(* PLC project RACK2537.project, Inovance company InoProShop(V1.8.1.3) InoProShop(V1.8.1.3) *)
(* stored: creationDateTime 2025-03-21T09:54:46.669365, modificationDateTime 2025-03-07T16:07:54.7010798 *)

TYPE _sDT : STRUCT
  year : DINT;  (* 按360天计算 *)
  month : DINT;  (* 按12个月计算 *)
  day : DINT;  (* 按30天计算 *)
  hour : DINT;  (* 按24小时 *)
  min : DINT;  (* 按60分钟 *)
  sec : DINT;  (* 按60秒 *)
END_STRUCT;
END_TYPE

FUNCTION_BLOCK 累计TIME
  VAR_INPUT
    EN : BOOL;
  END_VAR
  VAR
    心跳 : BOOL;
    TON_0 : TON;
    PLS_0 : PLS;
    TON_1 : TON;
  END_VAR
  VAR_INPUT
    清除 : BOOL;
  END_VAR
  VAR_OUTPUT
    ENO : BOOL;
    累计时间 : DINT;
  END_VAR
  VAR
    转换参数 : _sDT;
  END_VAR
  VAR_OUTPUT
    时间转换 : _sDT;
  END_VAR
  VAR  (* added by the conversion: wires and edge detectors of the diagram *)
    _GT49_ENO : BOOL;
    _GT49_OUT : BOOL;
  END_VAR

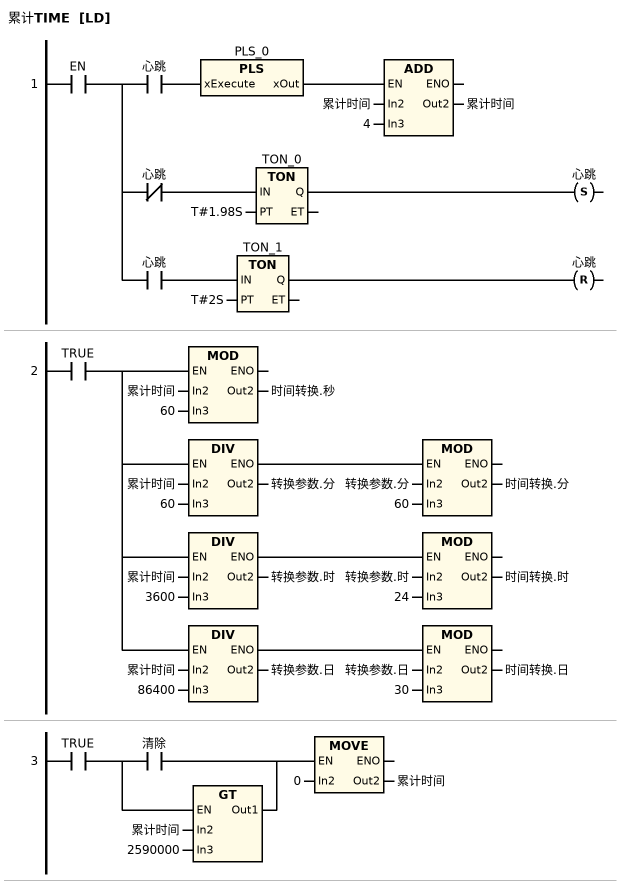
(* LD diagram, written out as Structured Text *)
(* 计时 *)

PLS_0(xExecute := EN AND 心跳);
IF PLS_0.xOut THEN 累计时间 := 累计时间 + 4; END_IF;
TON_0(IN := EN AND NOT 心跳, PT := T#1.98S);
IF TON_0.Q THEN 心跳 := TRUE; END_IF;
TON_1(IN := EN AND 心跳, PT := T#2S);
IF TON_1.Q THEN 心跳 := FALSE; END_IF;
(* 转换 *)

IF TRUE THEN 时间转换.秒 := 累计时间 MOD 60; END_IF;
IF TRUE THEN 转换参数.分 := 累计时间 / 60; END_IF;
IF TRUE THEN 时间转换.分 := 转换参数.分 MOD 60; END_IF;
IF TRUE THEN 转换参数.时 := 累计时间 / 3600; END_IF;
IF TRUE THEN 时间转换.时 := 转换参数.时 MOD 24; END_IF;
IF TRUE THEN 转换参数.日 := 累计时间 / 86400; END_IF;
IF TRUE THEN 时间转换.日 := 转换参数.日 MOD 30; END_IF;
(* 清除 *)

_GT49_OUT := GT(EN := TRUE, IN1 := 累计时间, IN2 := 2590000, ENO => _GT49_ENO);
IF TRUE AND 清除 OR _GT49_OUT THEN 累计时间 := 0; END_IF;
END_FUNCTION_BLOCK
